// TwinCAT 3 PLC project smallproject
// ProgramVersion: 3.1.4024.0
// libraries:
//   Tc2_Standard, * (Beckhoff Automation GmbH)
//   Tc2_System, * (Beckhoff Automation GmbH)
//   Tc3_Module, * (Beckhoff Automation GmbH)
// project tree:
//   Types/ ST_Sample.TcDUT
//   Globals/ GVL_Global.TcGVL
//   Programs/ Main.TcPOU
//   Tasks/ PlcTask.TcTTO
// real-time tasks:
//   TASK 2ms: cycle T#2ms, priority 3, ADS port 350
//   TASK 10ms: cycle T#10ms, priority 4, ADS port 351
//   TASK 200ms: cycle T#200000us, priority 6, ADS port 352
//   TASK FileWriterTask: cycle T#200000us, priority 1, ADS port 353
//   TASK PlcTask: cycle T#10ms, priority 20, ADS port 354
// I/O:
//   DEVICE Device 1 (EtherCAT) (disabled), AmsNetId 0.0.0.0.2.1
//     TermEtherCAT (EK1200) [EK1200-5000 EtherCAT Power supply (2A E-Bus)]
//       TermPower1 (EL9222-5500) [EL9222-5500 Overcurrent protection 24V DC, 2Ch., max. 10A (sum), adjustable]
//       TermOutput (EL2008) [EL2008 8Ch. Dig. Output 24V, 0.5A]
//       TermSensorGnrl (EL6224) [EL6224 (IO Link Master)]
//       TermPower2 (EL9222-5500) [EL9222-5500 Overcurrent protection 24V DC, 2Ch., max. 10A (sum), adjustable]
//       TermSensorFront (EL6224) [EL6224 (IO Link Master)]
//       TermSensorBack (EL6224) [EL6224 (IO Link Master)]
//       TermSensorEndstop (EL6224) [EL6224 (IO Link Master)]
//       Pr [EL6224 (IO Link Master)]
//       TermSafety (EL2911) [EL2911, Potential supply terminal (10 A) with 4 Ch. Safety Inputs, TwinSAFE]
//         modules: Module 2 (FSOUT), Module 3 (DEVICEIO), Module 4 (FSLOGIC)
//     Term 31 (EL3062) [EL3062 2Ch. Ana. Input 0-10V]
//     Term 32 (EL9505) [EL9505 Power supply terminal 5V]
//     Term 18 (EL9011) [EL9011 End Terminal]
//   DEVICE CanopenMaster (disabled), AmsNetId 0.0.0.0.6.1
//     DriveLnMn_15
//     Lift_18_Brake
//     DriveMain_17
//     DriveLane_16
//     Bms_32

CONFIGURATION smallproject
    RESOURCE PLC ON TwinCAT3
        TASK PlcTask(INTERVAL := T#10ms, PRIORITY := 20);
        PROGRAM Main WITH PlcTask : Main;
    END_RESOURCE
END_CONFIGURATION

// ---- Types/ST_Sample.TcDUT
TYPE ST_Sample :
STRUCT
	nCounter : INT;
	bReady : BOOL;
	aIntArray : ARRAY[0..50] OF INT;  
END_STRUCT
END_TYPE

// ---- Globals/GVL_Global.TcGVL
{attribute 'qualified_only'}
VAR_GLOBAL
	nMyInt : INT := 0;
	bMyBool : BOOL;
	nMyDint : DINT;

	nMyIntCounter : INT := 0;
	bMyBoolToogle : BOOL := FALSE;

	bIntCounterActive : BOOL := TRUE;
	bBoolToggleActive : BOOL := TRUE;

	// Period used by the timed logic (modifiable via ADS)
	tCyclePeriod : TIME := T#2S;

	// -----------------------

	nTimedIntCounter : INT := 0;
	bTimedBoolToogle : BOOL := FALSE;

	bTimedCounterActive : BOOL := TRUE;
	bTimedToggleActive : BOOL := TRUE;

	aIntArray : ARRAY[0..100] OF INT;  

	stMySampleStruct : ST_Sample;
	
	{attribute 'displaymode':='hex'}
	nVarWithStandardAttribute : DWORD;
	
	{attribute 'custom_attribute':='custom_attribute_value'}
	nVarWithCustomAttribute : DWORD;
END_VAR

// ---- Programs/Main.TcPOU
PROGRAM Main
VAR
	fbTimer : TON;
END_VAR

// ------------------------------------------------------------
// A) Cycle-based behavior (each PLC scan)
// ------------------------------------------------------------

IF GVL_Global.bIntCounterActive THEN
	GVL_Global.nMyIntCounter := GVL_Global.nMyIntCounter + 1;
END_IF

IF GVL_Global.bBoolToggleActive THEN
	GVL_Global.bMyBoolToogle := NOT GVL_Global.bMyBoolToogle;
END_IF

// ------------------------------------------------------------
// B) Time-based behavior (every tCyclePeriod)
// This triggers a "tick" each time the TON elapses.
// ------------------------------------------------------------
fbTimer(IN := TRUE, PT := GVL_Global.tCyclePeriod);

IF fbTimer.Q THEN
	// Do the same actions, but only on the tick
	IF GVL_Global.bTimedCounterActive THEN
		GVL_Global.nTimedIntCounter := GVL_Global.nTimedIntCounter + 1;
	END_IF
	
	IF GVL_Global.bTimedToggleActive THEN
		GVL_Global.bTimedBoolToogle := NOT GVL_Global.bTimedBoolToogle;
	END_IF
	
	// Retrigger timer (create a periodic pulse)
	fbTimer(IN := FALSE);
END_IF

END_PROGRAM
